TYPE ST_ManualMode :
STRUCT
	bKeyPos: BOOL;
	bKeyNeg: BOOL;
	bKeyRapid: BOOL;
	nLogAxisNumber: UINT;
	nInc: UDINT;
	nManualTyp: UINT;
	nSpeed: UINT;
	/// Handradauflösung in 0.1 um / Umdrehung 
	nHwResolution: UDINT;
END_STRUCT
END_TYPE

(* stored: Version 1.1.0.1, ProductVersion 3.1.4019.2
   DUT ST_ManualMode: Id {081593a3-81b6-48c8-ad5f-8ccfbc3cc3bd} *)
